// TIA Portal V19 export
VAR_GLOBAL   // PLC tag table "NEW INPUTS"
   "EMG STOP IP" AT %I0.0 : Bool;
   "PHASE FAIL IP" AT %I0.1 : Bool;
   "HOOTER RESET IP" AT %I0.2 : Bool;
   "AUTO/MAN SW IP" AT %I0.3 : Bool;
   "MGF FEED PUMP RUN IP" AT %I0.4 : Bool;
   "RO 1 HPP RUN IP" AT %I0.5 : Bool;
   "RO 2 HPP RUN IP" AT %I0.6 : Bool;
   "CIP PUMP RUN IP" AT %I0.7 : Bool;
   "PW TRANSFER PUMP - W RUN IP" AT %I1.0 : Bool;
   "PW TRANSFER PUMP - S RUN IP" AT %I1.1 : Bool;
   "PW TRANSFER W/P" AT %I1.2 : Bool;
   "AIR PRESSURE FAIL" AT %I1.3 : Bool;
   "SPARE IP3" AT %I1.4 : Bool;
   "LS-5 TANK LOW IP" AT %I1.5 : Bool;
   "LS-5 TANK HIGH IP" AT %I12.0 : Bool;
   "SPARE IP4" AT %I12.1 : Bool;
   "SPARE IP5" AT %I12.2 : Bool;
   "SPARE IP6" AT %I12.3 : Bool;
   "SPARE IP7" AT %I12.4 : Bool;
   "SPARE IP8" AT %I12.5 : Bool;
   "LPS-1" AT %I12.6 : Bool;
   "LPS-2" AT %I12.7 : Bool;
   "MGF V-1 OPEN FB" AT %I13.0 : Bool;
   "MGF V-2 OPEN FB" AT %I13.2 : Bool;
   "MGF V-3 OPEN FB" AT %I13.4 : Bool;
   "MGF V-4 OPEN FB" AT %I13.6 : Bool;
   "MGF V-1 CLOSE FB" AT %I13.1 : Bool;
   "MGF V-2 CLOSE FB" AT %I13.3 : Bool;
   "MGF V-3 CLOSE FB" AT %I13.5 : Bool;
   "MGF V-4 CLOSE FB" AT %I13.7 : Bool;
   "MGF V-5 OPEN FB" AT %I16.0 : Bool;
   "MGF V-5 CLOSE FB" AT %I16.1 : Bool;
   "ACF OPEN FB V1" AT %I16.2 : Bool;
   "ACF OPEN FB V2" AT %I16.4 : Bool;
   "ACF OPEN FB V3" AT %I16.6 : Bool;
   "ACF OPEN FB V4" AT %I17.0 : Bool;
   "ACF OPEN FB V5" AT %I17.2 : Bool;
   "ACF CLOSE FB V1" AT %I16.3 : Bool;
   "ACF CLOSE FB V2" AT %I16.5 : Bool;
   "ACF CLOSE FB V3" AT %I16.7 : Bool;
   "ACF CLOSE FB V4" AT %I17.1 : Bool;
   "ACF CLOSE FB V5" AT %I17.3 : Bool;
   "SF OPEN FB V1" AT %I17.4 : Bool;
   "SF OPEN FB V2" AT %I17.6 : Bool;
   "SF OPEN FB V3" AT %I20.0 : Bool;
   "SF OPEN FB V4" AT %I20.2 : Bool;
   "SF OPEN FB V5" AT %I20.4 : Bool;
   "SF OPEN FB V6" AT %I20.6 : Bool;
   "SF OPEN FB V7" AT %I21.0 : Bool;
   "SF CLOSE FB V1" AT %I17.5 : Bool;
   "SF CLOSE FB V2" AT %I17.7 : Bool;
   "SF CLOSE FB V3" AT %I20.1 : Bool;
   "SF CLOSE FB V4" AT %I20.3 : Bool;
   "SF CLOSE FB V5" AT %I20.5 : Bool;
   "SF CLOSE FB V6" AT %I20.7 : Bool;
   "SF CLOSE FB V7" AT %I21.1 : Bool;
   "SPARE IP9" AT %I21.2 : Bool;
   "SPARE IP10" AT %I21.3 : Bool;
   "SPARE IP11" AT %I21.4 : Bool;
   "SPARE IP12" AT %I21.5 : Bool;
   "SPARE IP13" AT %I21.6 : Bool;
   "SPARE IP14" AT %I21.7 : Bool;
END_VAR
